// TIA Portal V20 export
TYPE "LER_typeCmStatus"
// stored: Access Published
   STRUCT
      axisControl { ExternalWritable := 'False'} : Array[0..9] of "LBC_typeAxisControlNodeMonitoring";
      axis64Pos { ExternalWritable := 'False'} : Array[0..9] of "LBC_typeAxis64PosControlNodeMonitoring";
      sinaSpeed { ExternalWritable := 'False'} : Array[0..9] of "LBC_typeSinaSpeedControlNodeMonitoring";
      twoWayAct { ExternalWritable := 'False'} : Array[0..29] of "LBC_typeTwoWayActuatorControlNodeMonitoring";
      digitalSignal { ExternalWritable := 'False'} : Array[0..9] of "LBC_typeDigitalSignalControlNodeMonitoring";
      analogInput { ExternalWritable := 'False'} : Array[0..9] of "LBC_typeAnalogInputControlNodeMonitoring";
      analogOutput { ExternalWritable := 'False'} : Array[0..9] of "LBC_typeAnalogOutputControlNodeMonitoring";
   END_STRUCT;
END_TYPE
